FUNCTION_BLOCK FB_GetTemperature
VAR_INPUT
	terminalResistance : LREAL := 1;
	
	//values based on the EPCOS B57560G104F NTS sensor
	calibrationValues : ARRAY [1..6] OF LREAL := [25 ,100000 ,100 ,6338.3 , 200, 552.99];
	
END_VAR
VAR_OUTPUT
	temperatureSensor : LREAL;
END_VAR
VAR
	FBSteinHart : FB_SteinhartEquation; 
	A : LREAL;
	B : LREAL;
	C : LREAL;
END_VAR

// vraag steinhart parameters op
FBSteinHart(CV := calibrationValues , A => A, B => B, C => C);
// temperatuur wordt berekent met steainhart parameters en vergelijking
temperatureSensor := 1/(A+ B*LN(terminalResistance) + C * EXPT(LN(terminalResistance),3)); // steinhart equation is used to calculate the temperature of the sensor

END_FUNCTION_BLOCK

(* stored: Version 1.1.0.1, ProductVersion 3.1.4024.9
   POU FB_GetTemperature: Id {11c60e60-6f94-43ca-91bf-d0d09de39a4a}, SpecialFunc None *)
